FUNCTION_BLOCK ABSTRACT FB_ProfinetDevice EXTENDS FB_BaseDevice
VAR_INPUT
    // This is presented as a linkable input in the main project via a GVL
    StateInput AT %I* : UINT;
    // This is presented as a linkable input in the main project via a GVL
    DiagInput AT %I* : UINT;
	// This is presented as a linkable output in the main project via a GVL	
    CtrlOutput AT %Q* : UINT;
END_VAR
VAR
    uCtrlOutput : U_ProfinetDeviceCtrlOutput;
    uDiagInput  : U_ProfinetDeviceDiagInput;
    uStateInput : U_ProfinetDeviceStateInput;
END_VAR

END_FUNCTION_BLOCK

(* stored: Version 1.1.0.1, ProductVersion 3.1.4024.12
   POU FB_ProfinetDevice: Id {2509b0ae-d309-4bd3-86df-07912b9c1dea}, SpecialFunc None *)
